{attribute addProperty BoxType "EL1502--0000"}
{attribute addProperty Id "CNT_InputsAT %I*CNT_Inputs_2DD1A21088110CNT_OutputsAT %Q*CNT_Outputs_5A50AE9A6480WcStateAT %I*WcState_F855686C1620InfoDataAT %I*InfoData_BC63D37F80100"}
{attribute addProperty CRC "3224417886"}
{attribute addProperty SizeInBites "248"}
{attribute addProperty SizeInBytes "31"}
TYPE EL1502_D4B4E31B :
STRUCT
	{attribute addProperty Name "CNT_Inputs"}
	CNT_Inputs : CNT_Inputs_2DD1A210;
	{attribute addProperty Name "CNT_Outputs"}
	CNT_Outputs : CNT_Outputs_5A50AE9A;
	{attribute addProperty Name "WcState"}
	WcState : WcState_F855686C;
	{attribute addProperty Name "InfoData"}
	InfoData : InfoData_BC63D37F;
END_STRUCT
END_TYPE

(* stored: Version 1.2.0.0, ProductVersion 3.1.4024.9
   DUT EL1502_D4B4E31B: Id {ce60275e-9a1a-4650-9f83-a2c531fe4be0} *)
